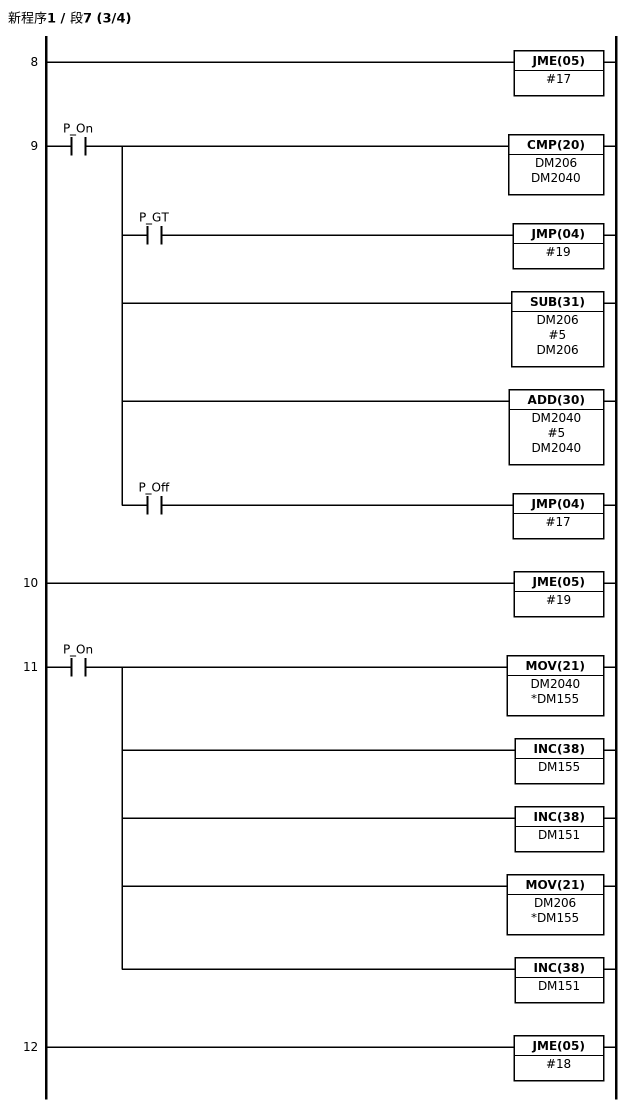
; [picture p24: 新程序1 / 段7, rungs 8-12]
; rung 8
JME(05) #17
; rung 9
LD P_On
OUT TR0
CMP(20) DM206 DM2040
AND P_GT
JMP(04) #19
LD TR0
SUB(31) DM206 #5 DM206
ADD(30) DM2040 #5 DM2040
AND P_Off
JMP(04) #17
; rung 10
JME(05) #19
; rung 11
LD P_On
MOV(21) DM2040 *DM155
INC(38) DM155
INC(38) DM151
MOV(21) DM206 *DM155
INC(38) DM151
; rung 12
JME(05) #18

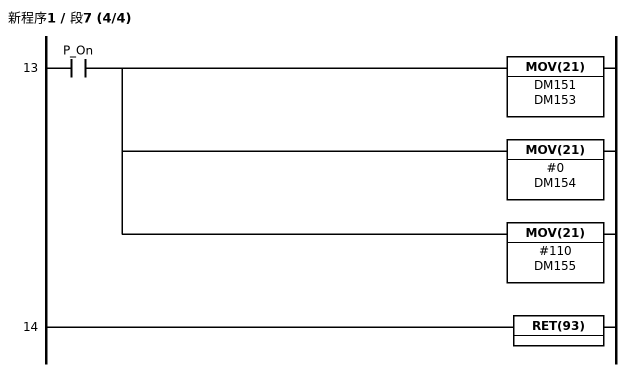
; rung 13
LD P_On
MOV(21) DM151 DM153
MOV(21) #0 DM154
MOV(21) #110 DM155
; rung 14
RET(93)

### Section 段8

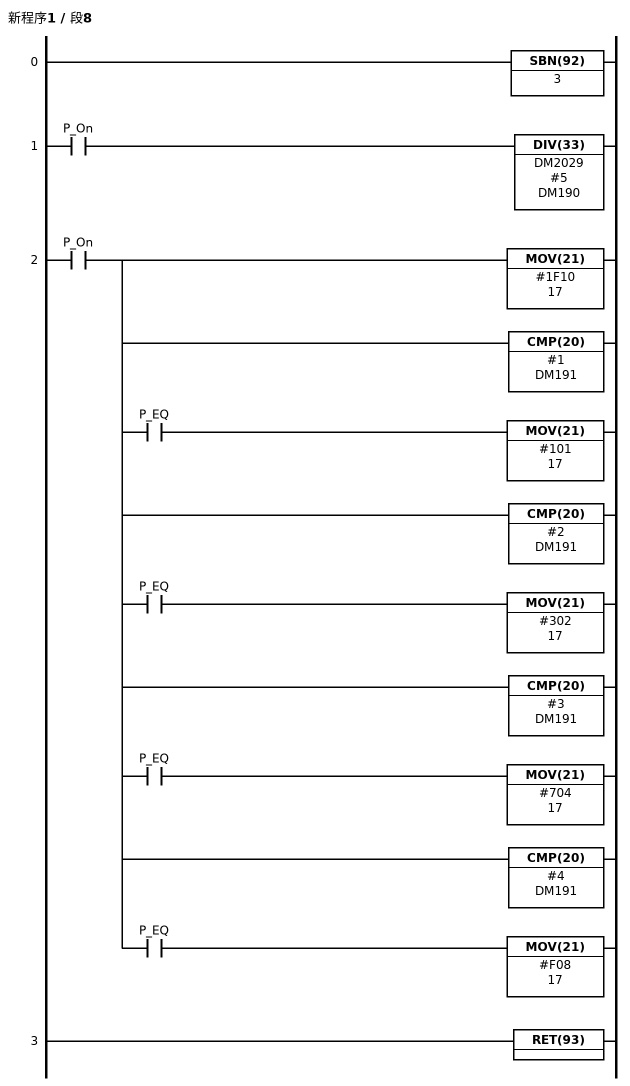
; rung 0
SBN(92) 3
; rung 1
LD P_On
DIV(33) DM2029 #5 DM190
; rung 2
LD P_On
OUT TR0
MOV(21) #1F10 17
CMP(20) #1 DM191
AND P_EQ
MOV(21) #101 17
LD TR0
CMP(20) #2 DM191
AND P_EQ
MOV(21) #302 17
LD TR0
CMP(20) #3 DM191
AND P_EQ
MOV(21) #704 17
LD TR0
CMP(20) #4 DM191
AND P_EQ
MOV(21) #F08 17
; rung 3
RET(93)

### Section 段9

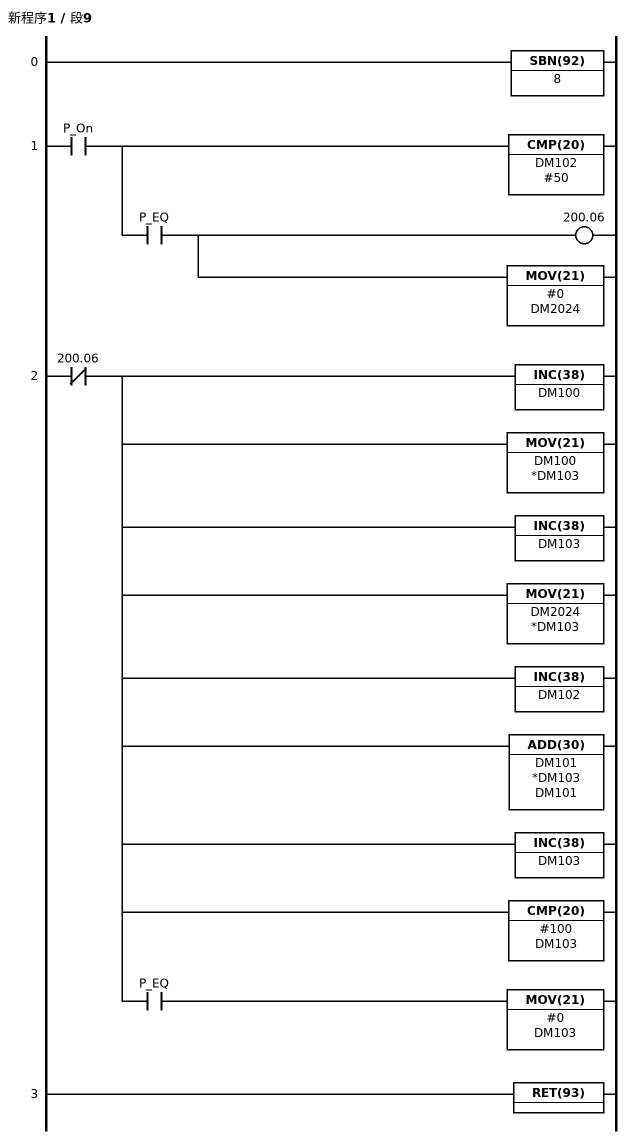
; rung 0
SBN(92) 8
; rung 1
LD P_On
CMP(20) DM102 #50
AND P_EQ
OUT 200.06
MOV(21) #0 DM2024
; rung 2
LDNOT 200.06
INC(38) DM100
MOV(21) DM100 *DM103
INC(38) DM103
MOV(21) DM2024 *DM103
INC(38) DM102
ADD(30) DM101 *DM103 DM101
INC(38) DM103
CMP(20) #100 DM103
AND P_EQ
MOV(21) #0 DM103
; rung 3
RET(93)

### Section 段10

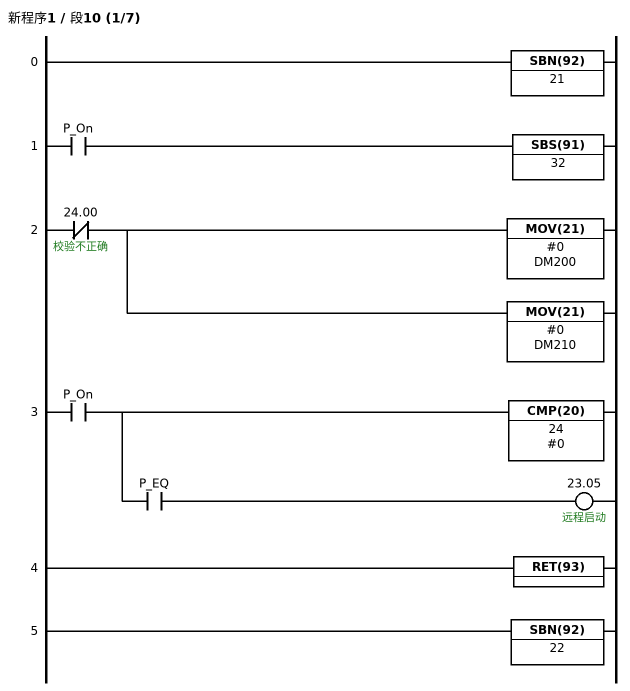
; rung 0
SBN(92) 21
; rung 1
LD P_On
SBS(91) 32
; rung 2
LDNOT 24.00  ; 校验不正确
MOV(21) #0 DM200
MOV(21) #0 DM210
; rung 3
LD P_On
CMP(20) 24 #0
AND P_EQ
OUT 23.05  ; 远程启动
; rung 4
RET(93)
; rung 5
SBN(92) 22

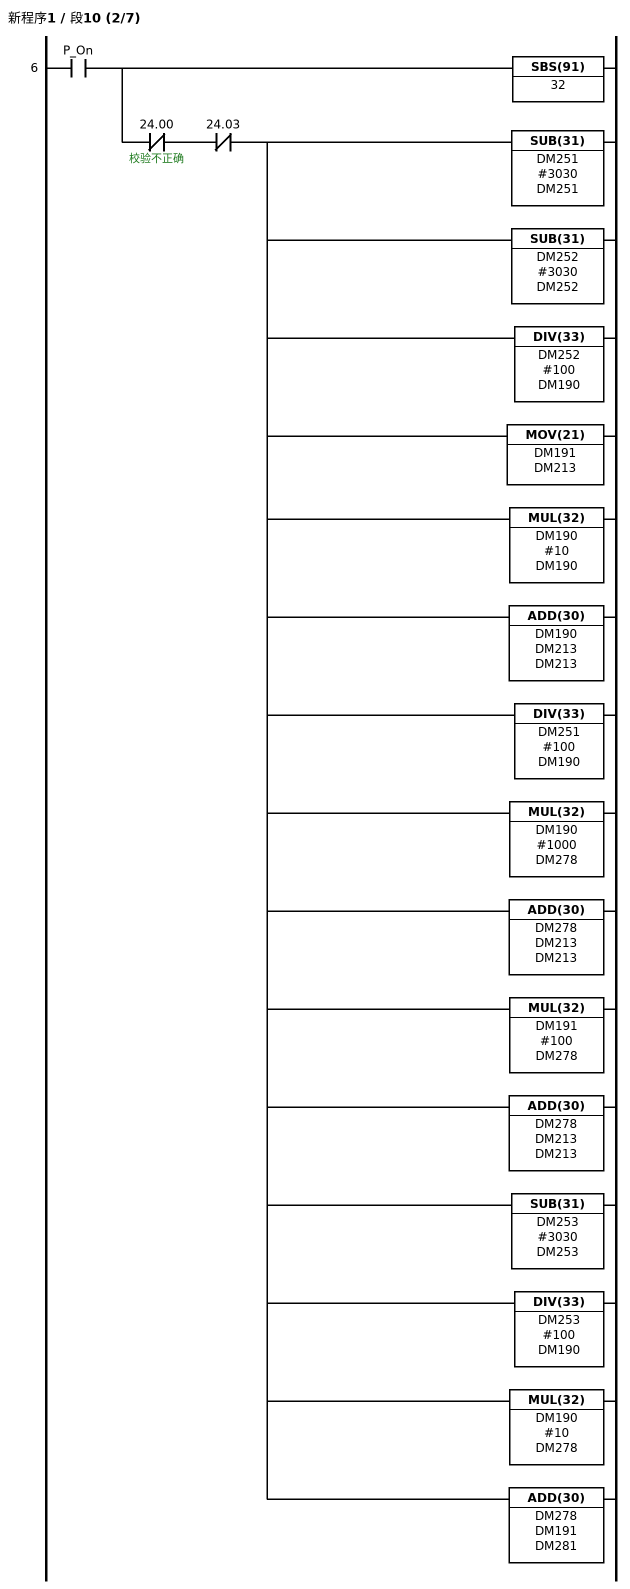
; rung 6
LD P_On
SBS(91) 32
ANDNOT 24.00  ; 校验不正确
ANDNOT 24.03
SUB(31) DM251 #3030 DM251
SUB(31) DM252 #3030 DM252
DIV(33) DM252 #100 DM190
MOV(21) DM191 DM213
MUL(32) DM190 #10 DM190
ADD(30) DM190 DM213 DM213
DIV(33) DM251 #100 DM190
MUL(32) DM190 #1000 DM278
ADD(30) DM278 DM213 DM213
MUL(32) DM191 #100 DM278
ADD(30) DM278 DM213 DM213
SUB(31) DM253 #3030 DM253
DIV(33) DM253 #100 DM190
MUL(32) DM190 #10 DM278
ADD(30) DM278 DM191 DM281

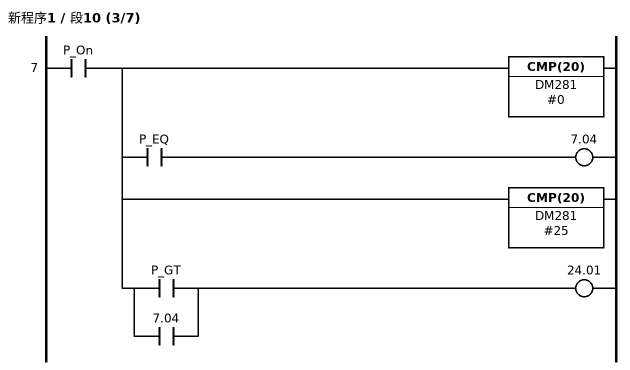
; rung 7
LD P_On
OUT TR0
CMP(20) DM281 #0
AND P_EQ
OUT 7.04
LD TR0
CMP(20) DM281 #25
LD P_GT
OR 7.04
ANDLD
OUT 24.01

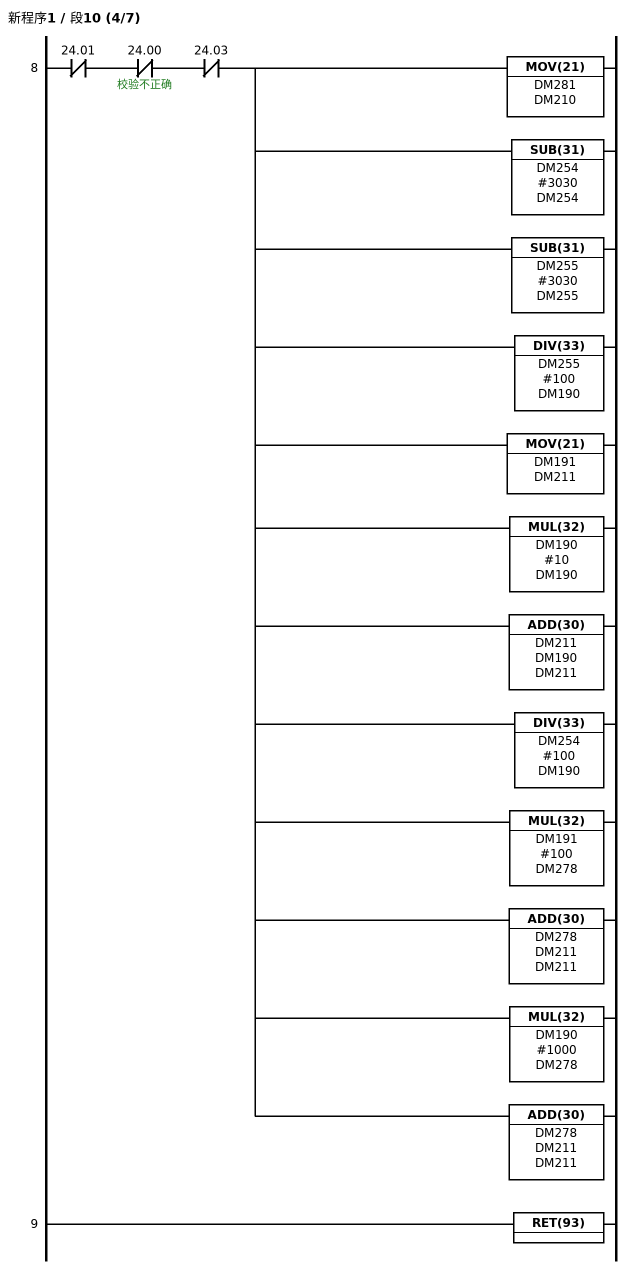
; rung 8
LDNOT 24.01
ANDNOT 24.00  ; 校验不正确
ANDNOT 24.03
MOV(21) DM281 DM210
SUB(31) DM254 #3030 DM254
SUB(31) DM255 #3030 DM255
DIV(33) DM255 #100 DM190
MOV(21) DM191 DM211
MUL(32) DM190 #10 DM190
ADD(30) DM211 DM190 DM211
DIV(33) DM254 #100 DM190
MUL(32) DM191 #100 DM278
ADD(30) DM278 DM211 DM211
MUL(32) DM190 #1000 DM278
ADD(30) DM278 DM211 DM211
; rung 9
RET(93)

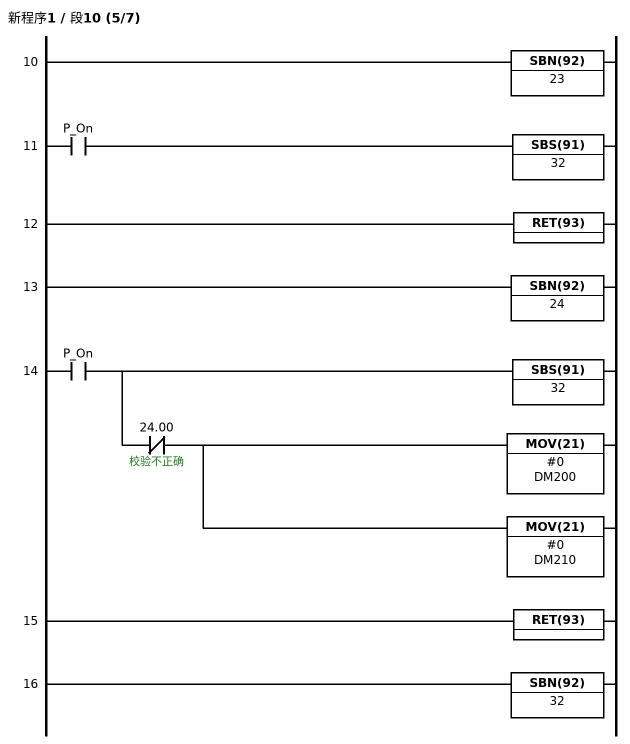
; rung 10
SBN(92) 23
; rung 11
LD P_On
SBS(91) 32
; rung 12
RET(93)
; rung 13
SBN(92) 24
; rung 14
LD P_On
SBS(91) 32
ANDNOT 24.00  ; 校验不正确
MOV(21) #0 DM200
MOV(21) #0 DM210
; rung 15
RET(93)
; rung 16
SBN(92) 32

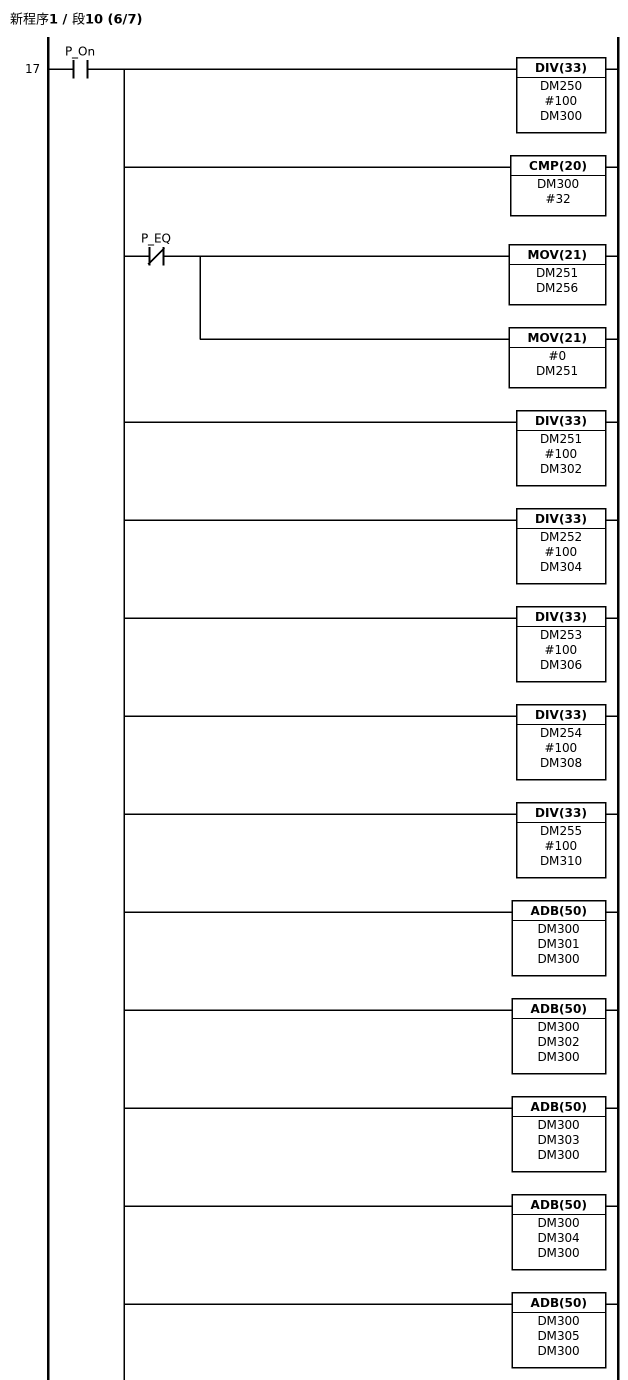

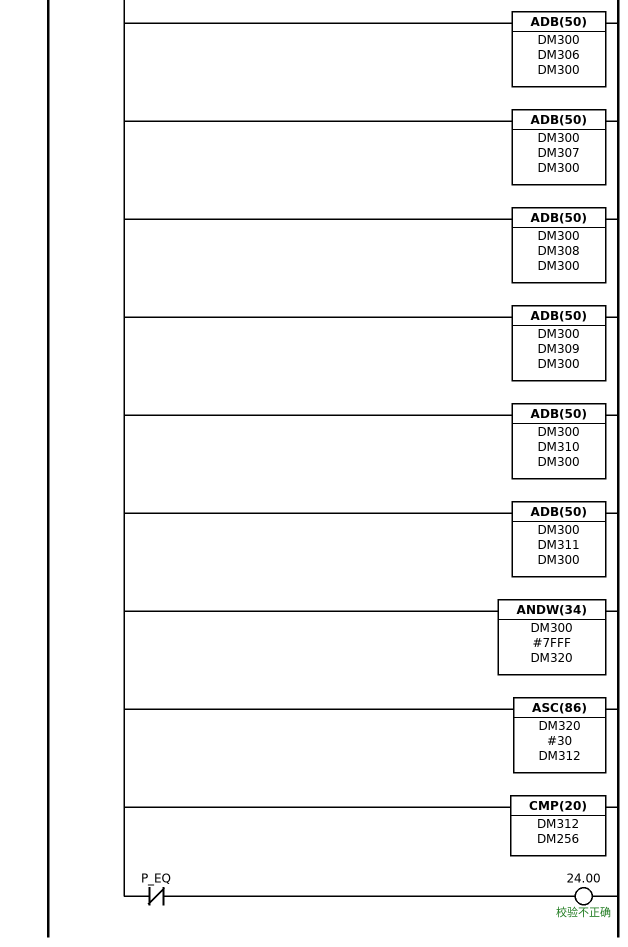
; rung 17
LD P_On
OUT TR0
DIV(33) DM250 #100 DM300
CMP(20) DM300 #32
ANDNOT P_EQ
MOV(21) DM251 DM256
MOV(21) #0 DM251
LD TR0
DIV(33) DM251 #100 DM302
DIV(33) DM252 #100 DM304
DIV(33) DM253 #100 DM306
DIV(33) DM254 #100 DM308
DIV(33) DM255 #100 DM310
ADB(50) DM300 DM301 DM300
ADB(50) DM300 DM302 DM300
ADB(50) DM300 DM303 DM300
ADB(50) DM300 DM304 DM300
ADB(50) DM300 DM305 DM300
ADB(50) DM300 DM306 DM300
ADB(50) DM300 DM307 DM300
ADB(50) DM300 DM308 DM300
ADB(50) DM300 DM309 DM300
ADB(50) DM300 DM310 DM300
ADB(50) DM300 DM311 DM300
ANDW(34) DM300 #7FFF DM320
ASC(86) DM320 #30 DM312
CMP(20) DM312 DM256
ANDNOT P_EQ
OUT 24.00  ; 校验不正确

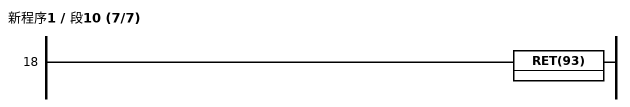
; rung 18
RET(93)

### Section 段11

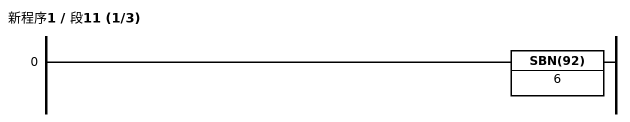
; rung 0
SBN(92) 6

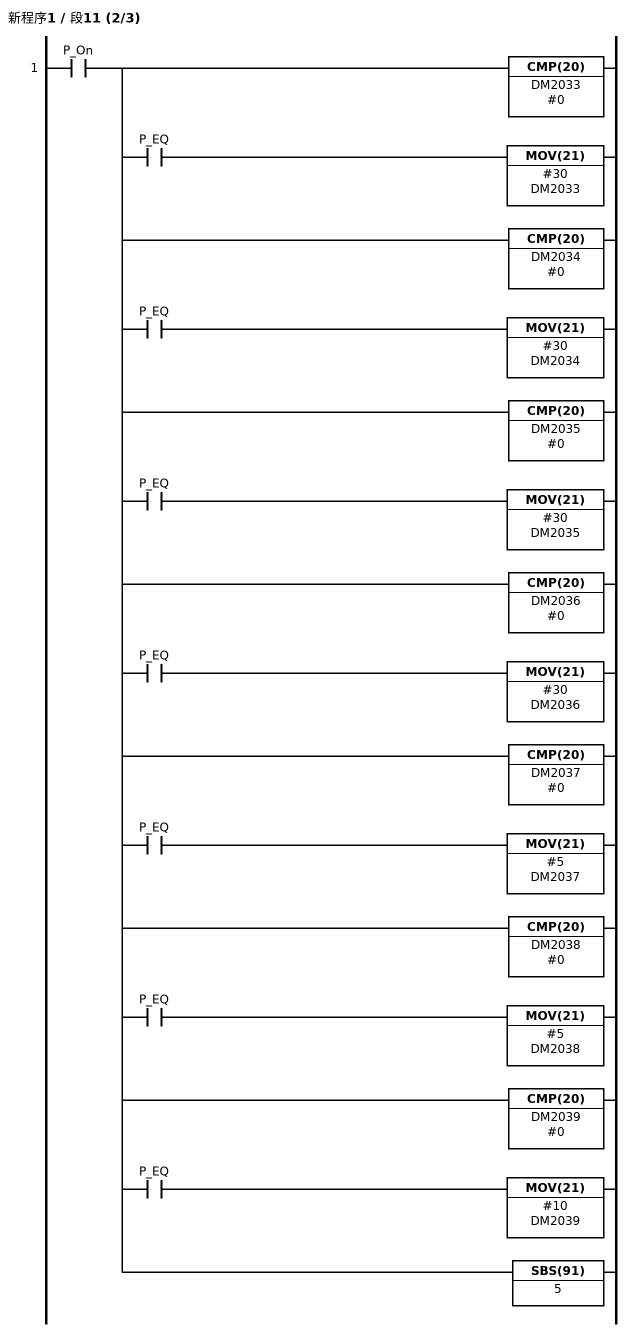
; rung 1
LD P_On
OUT TR0
CMP(20) DM2033 #0
AND P_EQ
MOV(21) #30 DM2033
LD TR0
CMP(20) DM2034 #0
AND P_EQ
MOV(21) #30 DM2034
LD TR0
CMP(20) DM2035 #0
AND P_EQ
MOV(21) #30 DM2035
LD TR0
CMP(20) DM2036 #0
AND P_EQ
MOV(21) #30 DM2036
LD TR0
CMP(20) DM2037 #0
AND P_EQ
MOV(21) #5 DM2037
LD TR0
CMP(20) DM2038 #0
AND P_EQ
MOV(21) #5 DM2038
LD TR0
CMP(20) DM2039 #0
AND P_EQ
MOV(21) #10 DM2039
LD TR0
SBS(91) 5

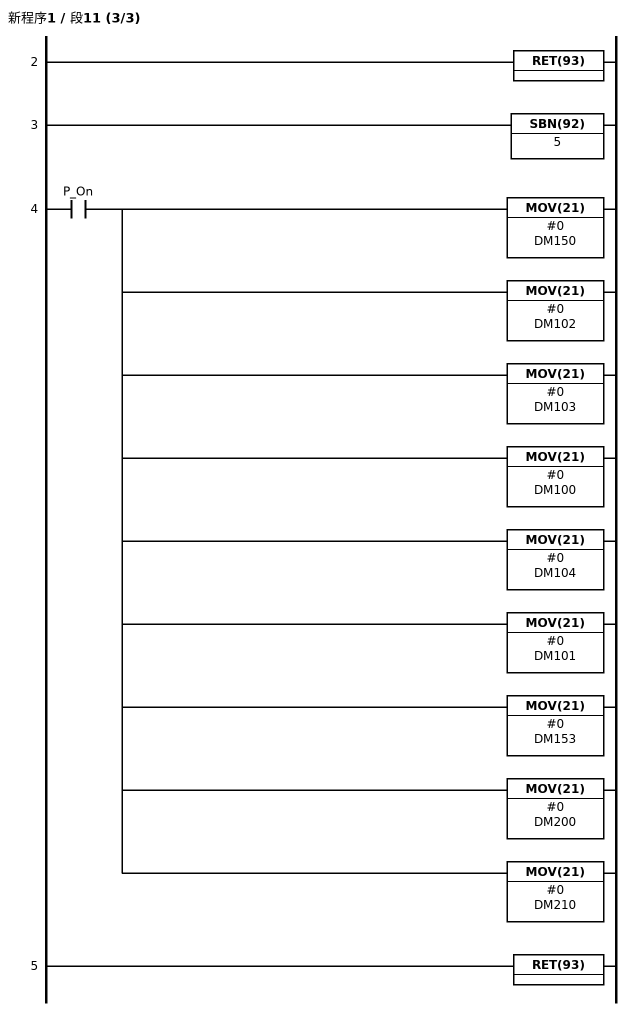
; rung 2
RET(93)
; rung 3
SBN(92) 5
; rung 4
LD P_On
MOV(21) #0 DM150
MOV(21) #0 DM102
MOV(21) #0 DM103
MOV(21) #0 DM100
MOV(21) #0 DM104
MOV(21) #0 DM101
MOV(21) #0 DM153
MOV(21) #0 DM200
MOV(21) #0 DM210
; rung 5
RET(93)

### Section 段12
; rung 0
END(01)